(* IEC 61131-3 sources: teller/JD_Teller_LC2_V11/Class/Call_JAM_Window, 1 file *)

(* ---- Call_JAM_Window.st ---- *)
(*!
<Class
	Name               = "Call_JAM_Window"
	Revision           = "1.0"
	RealtimeTask       = "false"
	CyclicTask         = "false"
	BackgroundTask     = "false"
	Sigmatek           = "false"
	OSInterface        = "false"
	HighPriority       = "false"
	Automatic          = "false"
	UpdateMode         = "Prescan"
	SharedCommandTable = "true"
	Objectsize         = "(630,120)">
	<Channels>
		<Server Name="ClassSvr" Visualized="true" Initialize="false" WriteProtected="false" Retentive="false"/>
	</Channels>
	<RevDoku>
		<Owner Company="JD"/>
		<Dokumentation Revision="1.0" Date="2014-10-29" Author="SV" Company="JD" Description=" SV client cJamLSE voor het tonen van het reset window in lse"/>
	</RevDoku>
</Class>
*)
Call_JAM_Window : CLASS
  //Servers:
	ClassSvr 	: SvrChCmd_DINT;
  //Clients:
  //Variables:
  //Functions:

	FUNCTION VIRTUAL GLOBAL ClassSvr::Write
		VAR_INPUT
			input (EAX) 	: DINT;
		END_VAR
		VAR_OUTPUT
			result (EAX) 	: DINT;
		END_VAR;
  //Tables:
	FUNCTION @STD
		VAR_OUTPUT
			ret_code	: CONFSTATES;
		END_VAR;
	FUNCTION GLOBAL TAB @CT_;
END_CLASS;

FUNCTION VIRTUAL GLOBAL Call_JAM_Window::ClassSvr::Write
	VAR_INPUT
		input (EAX) 	: DINT;
	END_VAR
	VAR_OUTPUT
		result (EAX) 	: DINT;
	END_VAR
  VAR
  	tmpno : udint;
    myList : _ANYLST;
  END_VAR

	ClassSvr := input;
  myList := FUNCTIONLST;

  case ClassSvr of

    // 0 : tmpno := get_no_by_label(p0:="Functienaam_in_LSE", x1:=myList, x2:=0);
    0 : tmpno := get_no_by_label(p0:="scr_Back", x1:=myList, x2:=0);

    1 : tmpno := get_no_by_label(p0:="wnd_JAMRESET", x1:=myList, x2:=0);

  end_case;

  if tmpno <> DEFSCOPE then
    InsertCmd(x0:=CMD_FUNCTIONBLOCK, x1:=tmpno$dint, x2:=0);
  end_if;
 	result := ClassSvr;

END_FUNCTION
